Staubli VAL3: cakajProgress.pgx

program cakajProgress(num x_nCas)
  local num l_nNuml_nStartTime
  local num l_nTimeRazlika
  local num l_nStartTime
begin
  // cakajProgress
  // @param x_nCas(num)  Funkcija resetira progress bar in s pomocjo razlike
  // casa prek clock() funkcije steje koliko casa je preostalo do konca, medtem ko
  // posodablja progress bar (nProgress) na grafičnem vmesniku

  // Resetiraj progress display
  nProgress = 0
  // Postavi casovno razliko na 0
  l_nTimeRazlika = 0
  // Trenutno pretekle sekunde
  l_nStartTime = clock()
  while l_nTimeRazlika < x_nCas
    delay(0.1)
    l_nTimeRazlika = clock() - l_nStartTime
    nProgress = min(100*l_nTimeRazlika/x_nCas, 100)
  endWhile
end
